TYPE stErrorHistoryRow :
STRUCT
	tTimeStamp			: TIME;
	sDescription		: STRING(80);
	iWorkStep1			: INT;
	iWorkStep2			: INT;
	udiErrorCode		: UDINT; 
END_STRUCT
END_TYPE

(* stored: Version 1.1.0.1, ProductVersion 3.1.4024.15
   DUT stErrorHistoryRow: Id {31753d45-ddb0-4bff-b337-bbf2e937983b} *)
